FUNCTION_BLOCK FB_NCMotionStage EXTENDS FB_BaseMotionStage
VAR_INPUT
END_VAR
VAR_OUTPUT
END_VAR
VAR
END_VAR

{warning 'Add method implementation '}
METHOD CalibrateEncoderValue
END_METHOD

{warning 'Add method implementation '}
METHOD DriveVirtual
END_METHOD

{warning 'Add method implementation '}
METHOD ExposeNCParams
END_METHOD

{warning 'Add method implementation '}
METHOD Homing
END_METHOD

{warning 'Add method implementation '}
METHOD LogErrors
END_METHOD

{warning 'Add property implementation'}
PROPERTY LogMessage : STRING
GET
END_GET
SET
END_SET
END_PROPERTY

END_FUNCTION_BLOCK

(* stored: Version 1.1.0.1
   POU FB_NCMotionStage: Id {b66d51f3-ef40-4af4-a6c8-0da9aa527c2a}, SpecialFunc None
   Method CalibrateEncoderValue: Id {9b9aed7e-e6bb-4487-b4fd-8a86aa7c3cf0}
   Method DriveVirtual: Id {c716eeb1-e0de-4e6d-8f54-915a4945ea5c}
   Method ExposeNCParams: Id {7e9b86fb-9b06-4fb3-b22e-88cf58ff0498}
   Method Homing: Id {b7dcd97f-bebf-424a-ad9e-c3f27769a66e}
   Method LogErrors: Id {a3021d3d-9a5e-484a-8b92-120cf37c2697}
   Property LogMessage: Id {f8247b3d-235f-48de-bb42-1fb526346d1f}
   Get Get: Id {83601d44-756a-4d0d-9793-c673d51acc75}
   Set Set: Id {d928898b-1d19-41af-8916-8780088f790c} *)
